(* IEC 61131-3 sources: RL_MAR/experiments/comparison/llm4plc/results/deepseek-ai-DeepSeek-V3.2_20260506_104945/20260506_112539, 3 files *)

(* ---- generated_code_iteration_0.st ---- *)
START_ST

FUNCTION_BLOCK FB_SplitNumber
VAR_INPUT
    InputNumber : INT;
END_VAR
VAR_OUTPUT
    Thousands : INT;
    Hundreds : INT;
    Tens : INT;
    Ones : INT;
    Min : INT;
    error : BOOL;
    status : WORD;
END_VAR
VAR
    state : INT;
    prevState : INT;
    tempNumber : INT;
    minValue : INT;
END_VAR

CASE state OF
    0: (* STATE 0: INITIALIZE AND VALIDATE INPUT *)
        (* Reset all output variables *)
        Thousands := 0;
        Hundreds := 0;
        Tens := 0;
        Ones := 0;
        Min := 0;
        error := FALSE;
        status := 16#0000;
        (* Validate InputNumber range *)
        IF (InputNumber >= 0) AND (InputNumber <= 9999) THEN
            state := 1; (* Transition to STATE 1 *)
        ELSE
            state := 3; (* Transition to STATE 3 *)
        END_IF;

    1: (* STATE 1: SEPARATE DIGITS *)
        (* Calculate digit values using division and modulo *)
        Thousands := InputNumber / 1000;
        Hundreds := (InputNumber MOD 1000) / 100;
        Tens := (InputNumber MOD 100) / 10;
        Ones := InputNumber MOD 10;
        state := 2; (* Transition to STATE 2 *)

    2: (* STATE 2: FIND MINIMUM NON-ZERO DIGIT *)
        (* Initialize minValue to maximum INT *)
        minValue := 32767;
        (* Check Thousands digit *)
        IF Thousands <> 0 THEN
            minValue := minimal(minValue, Thousands);
        END_IF;
        (* Check Hundreds digit *)
        IF Hundreds <> 0 THEN
            minValue := minimal(minValue, Hundreds);
        END_IF;
        (* Check Tens digit *)
        IF Tens <> 0 THEN
            minValue := minimal(minValue, Tens);
        END_IF;
        (* Check Ones digit *)
        IF Ones <> 0 THEN
            minValue := minimal(minValue, Ones);
        END_IF;
        (* Determine Min output *)
        IF minValue = 32767 THEN
            Min := 0; (* All digits were zero *)
        ELSE
            Min := minValue;
        END_IF;
        state := 0; (* Transition back to STATE 0 for next cycle *)

    3: (* STATE 3: ERROR HANDLING *)
        (* Set error outputs *)
        error := TRUE;
        status := 16#8001;
        (* Zero all digit outputs *)
        Thousands := 0;
        Hundreds := 0;
        Tens := 0;
        Ones := 0;
        Min := 0;
        state := 0; (* Transition back to STATE 0 for next cycle *)

    ELSE
        (* Default case: reset to STATE 0 *)
        state := 0;
END_CASE;

(* Store current state for tracking if needed *)
prevState := state;

END_FUNCTION_BLOCK

END_ST

(* ---- generated_code_iteration_1.st ---- *)
START_REASON
The validation feedback indicates a CODESYS compiler error: "发现非预期的记号'Min'". This translates to "unexpected token 'Min'". In the provided ST code, "Min" is used as an output variable name. In CODESYS, "MIN" is a reserved keyword (a standard function for finding the minimum of two values). Using "Min" as a variable name conflicts with this reserved keyword, causing the compiler error. The solution is to rename the output variable to something that is not a reserved keyword, such as "MinDigit" or "MinNonZero". I will rename it to "MinDigit" for clarity. Additionally, I should ensure that the variable names are consistent throughout the code, including in the state machine logic and output assignments. No other syntax errors were reported, so only this renaming is required.
END_REASON

START_ST

FUNCTION_BLOCK FB_SplitNumber
VAR_INPUT
    InputNumber : INT;
END_VAR
VAR_OUTPUT
    Thousands : INT;
    Hundreds : INT;
    Tens : INT;
    Ones : INT;
    MinDigit : INT;
    error : BOOL;
    status : WORD;
END_VAR
VAR
    state : INT;
    prevState : INT;
    tempNumber : INT;
    minValue : INT;
END_VAR

CASE state OF
    0: (* STATE 0: INITIALIZE AND VALIDATE INPUT *)
        (* Reset all output variables *)
        Thousands := 0;
        Hundreds := 0;
        Tens := 0;
        Ones := 0;
        MinDigit := 0;
        error := FALSE;
        status := 16#0000;
        (* Validate InputNumber range *)
        IF (InputNumber >= 0) AND (InputNumber <= 9999) THEN
            state := 1; (* Transition to STATE 1 *)
        ELSE
            state := 3; (* Transition to STATE 3 *)
        END_IF;

    1: (* STATE 1: SEPARATE DIGITS *)
        (* Calculate digit values using division and modulo *)
        Thousands := InputNumber / 1000;
        Hundreds := (InputNumber MOD 1000) / 100;
        Tens := (InputNumber MOD 100) / 10;
        Ones := InputNumber MOD 10;
        state := 2; (* Transition to STATE 2 *)

    2: (* STATE 2: FIND MINIMUM NON-ZERO DIGIT *)
        (* Initialize minValue to maximum INT *)
        minValue := 32767;
        (* Check Thousands digit *)
        IF Thousands <> 0 THEN
            minValue := MIN(minValue, Thousands);
        END_IF;
        (* Check Hundreds digit *)
        IF Hundreds <> 0 THEN
            minValue := MIN(minValue, Hundreds);
        END_IF;
        (* Check Tens digit *)
        IF Tens <> 0 THEN
            minValue := MIN(minValue, Tens);
        END_IF;
        (* Check Ones digit *)
        IF Ones <> 0 THEN
            minValue := MIN(minValue, Ones);
        END_IF;
        (* Determine MinDigit output *)
        IF minValue = 32767 THEN
            MinDigit := 0; (* All digits were zero *)
        ELSE
            MinDigit := minValue;
        END_IF;
        state := 0; (* Transition back to STATE 0 for next cycle *)

    3: (* STATE 3: ERROR HANDLING *)
        (* Set error outputs *)
        error := TRUE;
        status := 16#8001;
        (* Zero all digit outputs *)
        Thousands := 0;
        Hundreds := 0;
        Tens := 0;
        Ones := 0;
        MinDigit := 0;
        state := 0; (* Transition back to STATE 0 for next cycle *)

    ELSE
        (* Default case: reset to STATE 0 *)
        state := 0;
END_CASE;

(* Store current state for tracking if needed *)
prevState := state;

END_FUNCTION_BLOCK

END_ST

(* ---- generated_code_iteration_2.st ---- *)
START_REASON
The validation feedback indicates an encoding issue: "ANTLR syntax check failed: 'gbk' codec can't decode byte 0xa2 in position 85: illegal multibyte sequence". This error typically occurs when non-ASCII characters (like special quotes or symbols) are present in the code. In the previous ST code, I used parentheses with asterisks for comments (e.g., "(* STATE 0: INITIALIZE AND VALIDATE INPUT *)"), which are standard in ST and should not cause encoding issues. However, the error message suggests a byte sequence that cannot be decoded with the 'gbk' codec, possibly due to invisible or special characters introduced during copy-pasting or generation. To resolve this, I will ensure the code contains only ASCII characters by removing any non-ASCII elements, such as curly quotes or special symbols, and verify comment formatting. I will rewrite the code from scratch using plain ASCII characters, ensuring all comments use standard "(*" and "*)" delimiters without any hidden special characters. Additionally, I will maintain the previous fix for renaming "Min" to "MinDigit" to avoid reserved keyword conflicts. No other syntax errors were reported, so focusing on encoding should resolve the issue.
END_REASON

START_ST

FUNCTION_BLOCK FB_SplitNumber
VAR_INPUT
    InputNumber : INT;
END_VAR
VAR_OUTPUT
    Thousands : INT;
    Hundreds : INT;
    Tens : INT;
    Ones : INT;
    MinDigit : INT;
    error : BOOL;
    status : WORD;
END_VAR
VAR
    state : INT;
    prevState : INT;
    tempNumber : INT;
    minValue : INT;
END_VAR

CASE state OF
    0:
        Thousands := 0;
        Hundreds := 0;
        Tens := 0;
        Ones := 0;
        MinDigit := 0;
        error := FALSE;
        status := 16#0000;
        IF (InputNumber >= 0) AND (InputNumber <= 9999) THEN
            state := 1;
        ELSE
            state := 3;
        END_IF;

    1:
        Thousands := InputNumber / 1000;
        Hundreds := (InputNumber MOD 1000) / 100;
        Tens := (InputNumber MOD 100) / 10;
        Ones := InputNumber MOD 10;
        state := 2;

    2:
        minValue := 32767;
        IF Thousands <> 0 THEN
            minValue := MIN(minValue, Thousands);
        END_IF;
        IF Hundreds <> 0 THEN
            minValue := MIN(minValue, Hundreds);
        END_IF;
        IF Tens <> 0 THEN
            minValue := MIN(minValue, Tens);
        END_IF;
        IF Ones <> 0 THEN
            minValue := MIN(minValue, Ones);
        END_IF;
        IF minValue = 32767 THEN
            MinDigit := 0;
        ELSE
            MinDigit := minValue;
        END_IF;
        state := 0;

    3:
        error := TRUE;
        status := 16#8001;
        Thousands := 0;
        Hundreds := 0;
        Tens := 0;
        Ones := 0;
        MinDigit := 0;
        state := 0;

    ELSE
        state := 0;
END_CASE;

prevState := state;

END_FUNCTION_BLOCK

END_ST
